// TIA Portal project "AWL LIBRO 5" (V11)

(* hardware
DEVICE "S7300/ET200 station_1"  SIMATIC 300-Station
   slot 0: "Perfil soporte_0"  Rail  6ES7 390-1***0-0AA0
   slot 2: "PLC_1"  CPU 313C-2 DP  6ES7 313-6CF03-0AB0  V2.6
      slot 0: "Interfaz MPI_1"  MPI
      slot 1: "Interfaz DP_1"  DP
      slot 2: "DI16/DO16_1"  DI16/DO16
      slot 4: "Contaje_1"  Counter
*)

// ===== PLC "PLC_1"  CPU 313C-2 DP =====

VAR_GLOBAL   // PLC tag table "Tabla de variables estándar"
   "PULSADOR" AT %I0.0 : Bool;
   "FC CIERRE" AT %I0.1 : Bool;
   "FC APERTURA" AT %I0.2 : Bool;
   "M1 SUBIDA" AT %A0.0 : Bool;
   "M1 BAJADA" AT %A0.1 : Bool;
   "SALIDAS" AT %AB0 : Byte;
   "CONTROL" AT %MB1 : Byte;
   "CONTROL SUBIDA" AT %M1.0 : Bool;
   "CONTROL BAJADA" AT %M1.1 : Bool;
   "F0" AT %M0.0 : Bool;
   "F1" AT %M0.1 : Bool;
   "F2" AT %M0.2 : Bool;
   "F3" AT %M0.3 : Bool;
   "F4" AT %M0.4 : Bool;
   "F5" AT %M0.5 : Bool;
   "CONTADOR" AT %MW10 : Int;
   "F6" AT %M0.6 : Bool;
   "F7" AT %M0.7 : Bool;
   "INVERSOR BAJADA Y A T0 SUBIDA" AT %M1.2 : Bool;
   "INVERSOR SUBIDA Y A T1 BAJADA" AT %M1.3 : Bool;
   "RESET C. S." AT %M1.4 : Bool;
   "RESET C. B." AT %M1.5 : Bool;
   "F8" AT %M2.0 : Bool;
   "T0" AT %T0 : Timer;
   "T1" AT %T1 : Timer;
   "T2" AT %T3 : Timer;
END_VAR

ORGANIZATION_BLOCK "Main"   // OB1, STL
TITLE = EJERICICO 5 . / "Main Program Sweep (Cycle)"
{ S7_Optimized_Access := 'FALSE' }
VERSION : 0.1
   VAR_TEMP
      OB1_EV_CLASS : Byte;   // Bits 0-3 = 1 (Coming event), Bits 4-7 = 1 (Event class 1)
      OB1_SCAN_1 : Byte;   // 1 (Cold restart scan 1 of OB 1), 3 (Scan 2-n of OB 1)
      OB1_PRIORITY : Byte;   // Priority of OB Execution
      OB1_OB_NUMBR : Byte;   // 1 (Organization block 1, OB1)
      OB1_RESERVED_1 : Byte;   // Reserved for system
      OB1_RESERVED_2 : Byte;   // Reserved for system
      OB1_PREV_CYCLE : Int;   // Cycle time of previous OB1 scan (milliseconds)
      OB1_MIN_CYCLE : Int;   // Minimum cycle time of OB1 (milliseconds)
      OB1_MAX_CYCLE : Int;   // Maximum cycle time of OB1 (milliseconds)
      OB1_DATE_TIME : Date_And_Time;   // Date and time OB1 started
   END_VAR
BEGIN
END_ORGANIZATION_BLOCK